{region '#Template'}
	{attribute 'Category' := 'General'}
	{attribute 'Version' := '0.0.1.0'}
	{attribute 'Tags' := 'General, Cabinet, Control cabinet, Event groups, Categories, Notification classes, Event classes'}
	{attribute 'Description' := 'Ereignisgruppen, Kategorien	// Event groups, categories'}
{endregion}
FUNCTION_BLOCK FB_BA_EvtGroups EXTENDS FB_BA_View
VAR_INPUT CONSTANT
	LifeSafety						: FB_BA_EvtCategory_SimpStandExt;
	AlarmTechnical					: FB_BA_EvtCategory_SimpStandExt;
	Disturbance						: FB_BA_EvtCategory_SimpStandExt;
	Maintenance						: FB_BA_EvtCategory_SimpStandExt;
	Notification					: FB_BA_EvtCategory_SimpStand;
	Other							: FB_BA_EvtCategory_SimpStand;
END_VAR

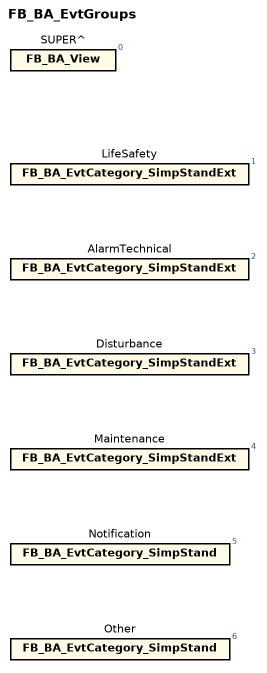
SUPER^(); // FB_BA_View
LifeSafety(); // FB_BA_EvtCategory_SimpStandExt
AlarmTechnical(); // FB_BA_EvtCategory_SimpStandExt
Disturbance(); // FB_BA_EvtCategory_SimpStandExt
Maintenance(); // FB_BA_EvtCategory_SimpStandExt
Notification(); // FB_BA_EvtCategory_SimpStand
Other(); // FB_BA_EvtCategory_SimpStand

METHOD FB_init : BOOL
VAR_INPUT
	bInitRetains : BOOL; // if TRUE, the retain variables are initialized (warm start / cold start)
	bInCopyCode : BOOL;  // if TRUE, the instance afterwards gets moved into the copy code (online change)
END_VAR
//===================================================================//
//	Life Safty
LifeSafety.iParent							:= THIS^;
LifeSafety.iLabel							:= LblCmpGeneral.EvtGroups_LifeSafety;									  
LifeSafety.sObjectName						:= '{Idx=01}';
LifeSafety.eDPADMode						:= E_BA_DPADMode.eInclude;																						
LifeSafety.Simple.nInstanceID				:= EventClasses.LifeSafetySimple;
LifeSafety.Simple.sObjectName				:= '{Idx=12}';
LifeSafety.Simple.eEventType				:= E_BA_EventType.eAlarm;
LifeSafety.Simple.eAlarmMode				:= E_BA_AlarmMode.eSimple;
LifeSafety.Simple.aPriority[1]				:= 10;
LifeSafety.Simple.aPriority[2]				:= 11;
LifeSafety.Simple.aPriority[3]				:= 12;
LifeSafety.Standard.nInstanceID				:= EventClasses.LifeSafetyStandard;
LifeSafety.Standard.sObjectName				:= '{Idx=11}';
LifeSafety.Standard.eEventType				:= E_BA_EventType.eAlarm;
LifeSafety.Standard.eAlarmMode				:= E_BA_AlarmMode.eStandard;
LifeSafety.Standard.aPriority[1]			:= 13;
LifeSafety.Standard.aPriority[2]			:= 14;
LifeSafety.Standard.aPriority[3]			:= 15;
LifeSafety.Extended.nInstanceID				:= EventClasses.LifeSafetyExtended;
LifeSafety.Extended.sObjectName				:= '{Idx=10}';
LifeSafety.Extended.eEventType				:= E_BA_EventType.eAlarm;
LifeSafety.Extended.eAlarmMode				:= E_BA_AlarmMode.eExtended;
LifeSafety.Extended.aPriority[1]			:= 16;
LifeSafety.Extended.aPriority[2]			:= 17;
LifeSafety.Extended.aPriority[3]			:= 18;

//===================================================================//
//	Alarm Technical
AlarmTechnical.iParent						:= THIS^;
AlarmTechnical.iLabel						:= LblCmpGeneral.EvtGroups_AlarmTechnical;									  
AlarmTechnical.sObjectName					:= '{Idx=01}';
AlarmTechnical.eDPADMode					:= E_BA_DPADMode.eInclude;																						
AlarmTechnical.Simple.nInstanceID			:= EventClasses.AlarmTechnicalSimple;
AlarmTechnical.Simple.sObjectName			:= '{Idx=22}';
AlarmTechnical.Simple.eEventType			:= E_BA_EventType.eAlarm;
AlarmTechnical.Simple.eAlarmMode			:= E_BA_AlarmMode.eSimple;
AlarmTechnical.Simple.aPriority[1]			:= 20;
AlarmTechnical.Simple.aPriority[2]			:= 21;
AlarmTechnical.Simple.aPriority[3]			:= 22;
AlarmTechnical.Standard.nInstanceID			:= EventClasses.AlarmTechnicalStandard;
AlarmTechnical.Standard.sObjectName			:= '{Idx=21}';
AlarmTechnical.Standard.eEventType			:= E_BA_EventType.eAlarm;
AlarmTechnical.Standard.eAlarmMode			:= E_BA_AlarmMode.eStandard;
AlarmTechnical.Standard.aPriority[1]		:= 23;
AlarmTechnical.Standard.aPriority[2]		:= 24;
AlarmTechnical.Standard.aPriority[3]		:= 25;
AlarmTechnical.Extended.nInstanceID			:= EventClasses.AlarmTechnicalExtended;
AlarmTechnical.Extended.sObjectName			:= '{Idx=20}';
AlarmTechnical.Extended.eEventType			:= E_BA_EventType.eAlarm;
AlarmTechnical.Extended.eAlarmMode			:= E_BA_AlarmMode.eExtended;
AlarmTechnical.Extended.aPriority[1]		:= 26;
AlarmTechnical.Extended.aPriority[2]		:= 27;
AlarmTechnical.Extended.aPriority[3]		:= 28;

//===================================================================//
//	Disturbance
Disturbance.iParent							:= THIS^;
Disturbance.iLabel							:= LblCmpGeneral.EvtGroups_Disturbance;									  
Disturbance.sObjectName						:= '{Idx=01}';
Disturbance.eDPADMode						:= E_BA_DPADMode.eInclude;																						
Disturbance.Simple.nInstanceID				:= EventClasses.DisturbanceSimple;
Disturbance.Simple.sObjectName				:= '{Idx=52}';
Disturbance.Simple.eEventType				:= E_BA_EventType.eAlarm;
Disturbance.Simple.eAlarmMode				:= E_BA_AlarmMode.eSimple;
Disturbance.Simple.aPriority[1]				:= 50;
Disturbance.Simple.aPriority[2]				:= 51;
Disturbance.Simple.aPriority[3]				:= 52;
Disturbance.Standard.nInstanceID			:= EventClasses.DisturbanceStandard;
Disturbance.Standard.sObjectName			:= '{Idx=51}';
Disturbance.Standard.eEventType				:= E_BA_EventType.eAlarm;
Disturbance.Standard.eAlarmMode				:= E_BA_AlarmMode.eStandard;
Disturbance.Standard.aPriority[1]			:= 53;
Disturbance.Standard.aPriority[2]			:= 54;
Disturbance.Standard.aPriority[3]			:= 55;
Disturbance.Extended.nInstanceID			:= EventClasses.DisturbanceExtended;
Disturbance.Extended.sObjectName			:= '{Idx=50}';
Disturbance.Extended.eEventType				:= E_BA_EventType.eAlarm;
Disturbance.Extended.eAlarmMode				:= E_BA_AlarmMode.eExtended;
Disturbance.Extended.aPriority[1]			:= 56;
Disturbance.Extended.aPriority[2]			:= 57;
Disturbance.Extended.aPriority[3]			:= 58;

//===================================================================//
//	Maintenance
Maintenance.iParent							:= THIS^;
Maintenance.iLabel							:= LblCmpGeneral.EvtGroups_Maintenance;									  
Maintenance.sObjectName						:= '{Idx=01}';
Maintenance.eDPADMode						:= E_BA_DPADMode.eInclude;																						
Maintenance.Simple.nInstanceID				:= EventClasses.MaintenanceSimple;
Maintenance.Simple.sObjectName				:= '{Idx=92}';
Maintenance.Simple.eEventType				:= E_BA_EventType.eAlarm;
Maintenance.Simple.eAlarmMode				:= E_BA_AlarmMode.eSimple;
Maintenance.Simple.aPriority[1]				:= 90;
Maintenance.Simple.aPriority[2]				:= 91;
Maintenance.Simple.aPriority[3]				:= 92;
Maintenance.Standard.nInstanceID			:= EventClasses.MaintenanceStandard;
Maintenance.Standard.sObjectName			:= '{Idx=91}';
Maintenance.Standard.eEventType				:= E_BA_EventType.eAlarm;
Maintenance.Standard.eAlarmMode				:= E_BA_AlarmMode.eStandard;
Maintenance.Standard.aPriority[1]			:= 93;
Maintenance.Standard.aPriority[2]			:= 94;
Maintenance.Standard.aPriority[3]			:= 95;
Maintenance.Extended.nInstanceID			:= EventClasses.MaintenanceExtended;
Maintenance.Extended.sObjectName			:= '{Idx=90}';
Maintenance.Extended.eEventType				:= E_BA_EventType.eAlarm;
Maintenance.Extended.eAlarmMode				:= E_BA_AlarmMode.eExtended;
Maintenance.Extended.aPriority[1]			:= 96;
Maintenance.Extended.aPriority[2]			:= 97;
Maintenance.Extended.aPriority[3]			:= 98;

//===================================================================//
//	Notification
Notification.iParent						:= THIS^;
Notification.iLabel							:= LblCmpGeneral.EvtGroups_Notification;									  
Notification.sObjectName					:= '{Idx=01}';
Notification.eDPADMode						:= E_BA_DPADMode.eInclude;																						
Notification.Simple.nInstanceID				:= EventClasses.NotificationSimple;
Notification.Simple.sObjectName				:= '{Idx=132}';
Notification.Simple.eEventType				:= E_BA_EventType.eAlarm;
Notification.Simple.eAlarmMode				:= E_BA_AlarmMode.eSimple;
Notification.Simple.aPriority[1]			:= 130;
Notification.Simple.aPriority[2]			:= 131;
Notification.Simple.aPriority[3]			:= 132;
Notification.Standard.nInstanceID			:= EventClasses.NotificationStandard;
Notification.Standard.sObjectName			:= '{Idx=131}';
Notification.Standard.eEventType			:= E_BA_EventType.eAlarm;
Notification.Standard.eAlarmMode			:= E_BA_AlarmMode.eStandard;
Notification.Standard.aPriority[1]			:= 133;
Notification.Standard.aPriority[2]			:= 134;
Notification.Standard.aPriority[3]			:= 135;

//===================================================================//
//	Other
Other.iParent								:= THIS^;
Other.iLabel								:= LblCmpGeneral.EvtGroups_Other;									  
Other.sObjectName							:= '{Idx=01}';
Other.eDPADMode								:= E_BA_DPADMode.eInclude;																						
Other.Simple.nInstanceID					:= EventClasses.OtherSimple;
Other.Simple.sObjectName					:= '{Idx=182}';
Other.Simple.eEventType						:= E_BA_EventType.eAlarm;
Other.Simple.eAlarmMode						:= E_BA_AlarmMode.eSimple;
Other.Simple.aPriority[1]					:= 180;
Other.Simple.aPriority[2]					:= 181;
Other.Simple.aPriority[3]					:= 182;
Other.Standard.nInstanceID					:= EventClasses.OtherStandard;
Other.Standard.sObjectName					:= '{Idx=181}';
Other.Standard.eEventType					:= E_BA_EventType.eAlarm;
Other.Standard.eAlarmMode					:= E_BA_AlarmMode.eStandard;
Other.Standard.aPriority[1]					:= 183;
Other.Standard.aPriority[2]					:= 184;
Other.Standard.aPriority[3]					:= 185;
END_METHOD

END_FUNCTION_BLOCK

(* stored: Version 1.1.0.1, ProductVersion 3.1.4024.6
   POU FB_BA_EvtGroups: Id {353e64f1-d0e6-4a29-a87b-7a0c4acab0df}, SpecialFunc None
   Method FB_init: Id {73c534cd-c339-4e66-944a-49dec33ce02a} *)
